	FUNCTION_BLOCK FB 1006
	TITLE =A_2111_MXZ41MA TRAVELING DRIVE
	//COPYRIGHT:     (C) 2009  BUHLER AG, CH-9240 UZWIL, SWITZERLAND
	//
	//PRODUCT:       WinCoS_BIW01_09
	//
	//TITLE:         TRAVELING DRIVE
	//
	//--------------------------------------------------------------------------------
	//
	//IDENT:         AUTHOR:             DEPT:                             DATE:
	//
	//P01_FB1006.1.0 K.Renz              CSB41                             12.Okt.2009
	//               1st Release
	//
	//--------------------------------------------------------------------------------
	//
	//PURPOSE:
	//
	//MANUAL :
	//
	//RESTRICTIONS:
	//
	//--------------------------------------------------------------------------------
	AUTHOR  : KR
	FAMILY  : USW
	VERSION : 0.0


	VAR
	         Ma :  UDT 20860  ;  // Machine
	         A_2111_MXZ41 : FB12;  // Motor: Motor
	         A_2111_MXZ41TF : FB17;  // AO Speed: AnaOutp
	         PLC1BIW01_02 : FB14; // LS Zero Position: DigInpCont
	         A_2111_MXZ41BLH : FB14; // LS Product Flow: DigInpCont
	         A_2111_MXZ41SM : FB14;  // SM: DigInpCont
	         IncCounter : UDT 20851;   // Counter module
	END_VAR

	BEGIN
	NETWORK
	TITLE =Call SSW
	   UC  FB86
	END_FUNCTION_BLOCK
